Yaskawa INFORM job: MCRSPD1.JBI

/JOB
//NAME MCRSPD1
//POS
///NPOS 0,0,0,0,0,0
//INST
///DATE 2010/10/22 12:49
///ATTR SC,RW,MC
///GROUP1 RB1
NOP
SKILLSND "spdoverride_on"
END
